FUNCTION_BLOCK FB_AlarmStatusManager
VAR_INPUT
    bMaintenanceMode : BOOL;  
END_VAR

VAR_OUTPUT
    stSystemStatus : ST_SystemAlarmStatus;  
END_VAR

VAR
    i : INT;
    bFirstRun : BOOL := TRUE;
    nZone : SINT;
    bIsGlobalAlarm : BOOL;
	
    aAllAlarms : ARRAY[1..100] OF ST_AlarmEntry;
    nAlarmCount : INT := 0;
	fbFlashTimer : TON;
	bFlashState  : BOOL;
END_VAR

stSystemStatus.bMaintenanceMode := bMaintenanceMode;

// Initialize alarm list 
IF bFirstRun THEN
    InitializeAlarmList();
    bFirstRun := FALSE;
END_IF

// Reset all zones to OK
bCriticalAlarm := FALSE;

FOR i := 1 TO 5 DO
    stSystemStatus.aZoneStatus[i].bOkToRun := TRUE;
    stSystemStatus.aZoneStatus[i].nHighestSeverity := 0;
END_FOR

//Check Safety Relay status
SafetyRelay.bCondition := NOT SafetyRelayStatus;

IF SafetyRelay.bCondition THEN
	(* Timer counts to 250ms, then resets itself *)
	fbFlashTimer(IN := NOT fbFlashTimer.Q, PT := T#250MS);

	(* Every time the timer finishes (Q=TRUE), toggle the state *)
	IF fbFlashTimer.Q THEN
		bFlashState := NOT bFlashState;
	END_IF

	(* Map to your physical output *)
	bResetLED := bFlashState;
ELSE
	bResetLED := FALSE;
END_IF

// Process all alarms 
FOR i := 1 TO nAlarmCount DO
    IF aAllAlarms[i].pAlarm <> 0 THEN
		nZone := ParseAlarmZone(aAllAlarms[i].sName);
		ProcessAlarm(aAllAlarms[i].pAlarm, nZone);	
    END_IF
	
END_FOR

METHOD AddAlarm : BOOL
VAR_INPUT
    pAlarm : POINTER TO ST_Alarm;
    sAlarmName : STRING(50);
END_VAR
nAlarmCount := nAlarmCount + 1;
aAllAlarms[nAlarmCount].pAlarm := pAlarm;
aAllAlarms[nAlarmCount].sName := sAlarmName;

AddAlarm := TRUE;
END_METHOD

METHOD InitializeAlarmList : BOOL
nAlarmCount := 0;

(* RAIL 1 *)
AddAlarm(ADR(GVL_Alarms.R1_Sensor_UnknownPosition), 'R1_Sensor_UnknownPosition');
AddAlarm(ADR(GVL_Alarms.R1_Sensor_MotionTimedOut), 'R1_Sensor_MotionTimedOut');
AddAlarm(ADR(GVL_Alarms.R1_Compressor_UnknownPosition), 'R1_Compressor_UnknownPosition');
AddAlarm(ADR(GVL_Alarms.R1_Compressor_MotionTimedOut), 'R1_Compressor_MotionTimedOut');
AddAlarm(ADR(GVL_Alarms.R1_Chariot_MotionTimedOut), 'R1_Chariot_MotionTimedOut');
AddAlarm(ADR(GVL_Alarms.R1_Chariot_UnknownPosition), 'R1_Chariot_UnknownPosition');
AddAlarm(ADR(GVL_Alarms.R1_Stepper_Motion_Failed), 'R1_Stepper_Motion_Failed');
AddAlarm(ADR(GVL_Alarms.R1_Stepper_Homing_Failed), 'R1_Stepper_Homing_Failed');
AddAlarm(ADR(GVL_Alarms.R1_Stepper_Motion_Interrupted), 'R1_Stepper_Motion_Interrupted');
AddAlarm(ADR(GVL_Alarms.R1_Stepper_PowerUp_Failed), 'R1_Stepper_PowerUp_Failed');
AddAlarm(ADR(GVL_Alarms.R1_Stepper_Reset_Failed), 'R1_Stepper_Reset_Failed');
AddAlarm(ADR(GVL_Alarms.R1_Stepper_Stop_Failed), 'R1_Stepper_Stop_Failed');
AddAlarm(ADR(GVL_Alarms.R1_Stepper_UnableToReadPosition), 'R1_Stepper_UnableToReadPosition');

(* RAIL 2 *)
AddAlarm(ADR(GVL_Alarms.R2_Stepper_PowerUp_Failed), 'R2_Stepper_PowerUp_Failed');
AddAlarm(ADR(GVL_Alarms.R2_Stepper_Homing_Failed), 'R2_Stepper_Homing_Failed');
AddAlarm(ADR(GVL_Alarms.R2_Stepper_Motion_Failed), 'R2_Stepper_Motion_Failed');
AddAlarm(ADR(GVL_Alarms.R2_Stepper_Motion_Interrupted), 'R2_Stepper_Motion_Interrupted');
AddAlarm(ADR(GVL_Alarms.R2_Stepper_Reset_Failed), 'R2_Stepper_Reset_Failed');
AddAlarm(ADR(GVL_Alarms.R2_Chariot_UnknownPosition), 'R2_Chariot_UnknownPosition');
AddAlarm(ADR(GVL_Alarms.R2_Chariot_MotionTimedOut), 'R2_Chariot_MotionTimedOut');
AddAlarm(ADR(GVL_Alarms.R2_Stepper_Stop_Failed), 'R2_Stepper_Stop_Failed');
AddAlarm(ADR(GVL_Alarms.R2_Stepper_UnableToReadPosition), 'R2_Stepper_UnableToReadPosition');

(* RAIL 3 *)
AddAlarm(ADR(GVL_Alarms.R3_Compressor_UnknownPosition), 'R3_Compressor_UnknownPosition');
AddAlarm(ADR(GVL_Alarms.R3_HeatExCoupola_DriveFaulted), 'R3_HeatExCoupola_DriveFaulted');
AddAlarm(ADR(GVL_Alarms.R3_RegenCoupola_DriveFaulted), 'R3_RegenCoupola_DriveFaulted');
AddAlarm(ADR(GVL_Alarms.R3_Compressor_MotionTimedOut), 'R3_Compressor_MotionTimedOut');
AddAlarm(ADR(GVL_Alarms.R3_HeatExCoupola_UnknownState), 'R3_HeatExCoupola_UnknownPosition');
AddAlarm(ADR(GVL_Alarms.R3_HeatExCoupola_MotionTimedOut), 'R3_HeatExCoupola_MotionTimedOut');
AddAlarm(ADR(GVL_Alarms.R3_RegenCoupola_UnknownPosition), 'R3_RegenCoupola_UnknownPosition');
AddAlarm(ADR(GVL_Alarms.R3_RegenCoupola_MotionTimedOut), 'R3_RegenCoupola_MotionTimedOut');
AddAlarm(ADR(GVL_Alarms.R3_Chariot_UnknownPosition), 'R3_Chariot_UnknownPosition');
AddAlarm(ADR(GVL_Alarms.R3_Chariot_MotionTimedOut), 'R3_Chariot_MotionTimedOut');
AddAlarm(ADR(GVL_Alarms.R3_Stepper_PowerUp_Failed), 'R3_Stepper_PowerUp_Failed');
AddAlarm(ADR(GVL_Alarms.R3_Stepper_Homing_Failed), 'R3_Stepper_Homing_Failed');
AddAlarm(ADR(GVL_Alarms.R3_Stepper_Motion_Failed), 'R3_Stepper_Motion_Failed');
AddAlarm(ADR(GVL_Alarms.R3_Stepper_Motion_Interrupted), 'R3_Stepper_Motion_Interrupted');
AddAlarm(ADR(GVL_Alarms.R3_Stepper_Reset_Failed), 'R3_Stepper_Reset_Failed');
AddAlarm(ADR(GVL_Alarms.R3_Stepper_Stop_Failed), 'R3_Stepper_Stop_Failed');
AddAlarm(ADR(GVL_Alarms.R3_Stepper_UnableToReadPosition), 'R3_Stepper_UnableToReadPosition');

(* RAIL 4 *)
AddAlarm(ADR(GVL_Alarms.R4_Stepper_PowerUp_Failed), 'R4_Stepper_PowerUp_Failed');
AddAlarm(ADR(GVL_Alarms.R4_Stepper_Homing_Failed), 'R4_Stepper_Homing_Failed');
AddAlarm(ADR(GVL_Alarms.R4_Stepper_Motion_Failed), 'R4_Stepper_Motion_Failed');
AddAlarm(ADR(GVL_Alarms.R4_Stepper_Motion_Interrupted), 'R4_Stepper_Motion_Interrupted');
AddAlarm(ADR(GVL_Alarms.R4_Stepper_Reset_Failed), 'R4_Stepper_Reset_Failed');
AddAlarm(ADR(GVL_Alarms.R4_Chariot_UnknownPosition), 'R4_Chariot_UnknownPosition');
AddAlarm(ADR(GVL_Alarms.R4_Chariot_MotionTimedOut), 'R4_Chariot_MotionTimedOut');
AddAlarm(ADR(GVL_Alarms.R4_Stepper_Stop_Failed), 'R4_Stepper_Stop_Failed');
AddAlarm(ADR(GVL_Alarms.R4_Stepper_UnableToReadPosition), 'R4_Stepper_UnableToReadPosition');

(* GLOBAL SECURITY *)
AddAlarm(ADR(GVL_Alarms.SafetyRelay), 'SafetyRelay');
InitializeAlarmList := TRUE;
END_METHOD

METHOD ParseAlarmZone : SINT
VAR_INPUT
    sAlarmName : STRING(50);
END_VAR
VAR
    sZoneChar : STRING(1);
    nZoneNum : SINT;
    sAfterR : STRING;
END_VAR
ParseAlarmZone := 0;

// Check if alarm is global or belongs to a zone
IF LEN(sAlarmName) >= 3 AND LEFT(sAlarmName, 1) = 'R' THEN

    sAfterR := RIGHT(sAlarmName, LEN(sAlarmName) - 1);
    
    sZoneChar := LEFT(sAfterR, 1);
    nZoneNum := STRING_TO_SINT(sZoneChar);
    
    IF nZoneNum >= 1 AND nZoneNum <= 4 AND LEFT(RIGHT(sAfterR, LEN(sAfterR) - 1), 1) = '_' THEN
        ParseAlarmZone := nZoneNum;
    END_IF
	
ELSE
    ParseAlarmZone := 5;  
END_IF
END_METHOD

METHOD ProcessAlarm : BOOL
VAR_INPUT
    pAlarm : POINTER TO ST_Alarm;
    nZone : SINT;
END_VAR
VAR
    nSeverity : UINT;
    bAlarmActive : BOOL;
END_VAR
// Check validity
IF pAlarm = 0 OR nZone < 1 OR nZone > 5 THEN
    ProcessAlarm := FALSE;
    RETURN;
END_IF

nSeverity := pAlarm^.nSeverity;
bAlarmActive := pAlarm^.bCondition;  

IF bAlarmActive THEN
    IF nSeverity > stSystemStatus.aZoneStatus[nZone].nHighestSeverity THEN
        stSystemStatus.aZoneStatus[nZone].nHighestSeverity := nSeverity;
    END_IF

    CASE nSeverity OF
        1, 2: // Info, Warning - No blocking 
            
        3, 4: // Error - Block unless maintenance mode
            IF NOT bMaintenanceMode THEN
                stSystemStatus.aZoneStatus[nZone].bOkToRun := FALSE;
            END_IF
            
        5: // Critical 
            stSystemStatus.aZoneStatus[nZone].bOkToRun := FALSE;
			bCriticalAlarm := TRUE;
    END_CASE
END_IF

ProcessAlarm := TRUE;
END_METHOD

END_FUNCTION_BLOCK

(* stored: Version 1.1.0.1, ProductVersion 3.1.4026.11
   POU FB_AlarmStatusManager: Id {05451d1b-b510-43ab-83d4-ae190ad58e7b}, SpecialFunc None
   Method AddAlarm: Id {6fdebe5e-54bc-4f7a-9386-b1b99075ac08}
   Method InitializeAlarmList: Id {29d25a2e-365e-4965-b599-96f6962c9be3}
   Method ParseAlarmZone: Id {40233a2f-1b32-4819-9f83-62c231758972}
   Method ProcessAlarm: Id {2dfd239b-192b-4991-b143-7c60f3898bff} *)
